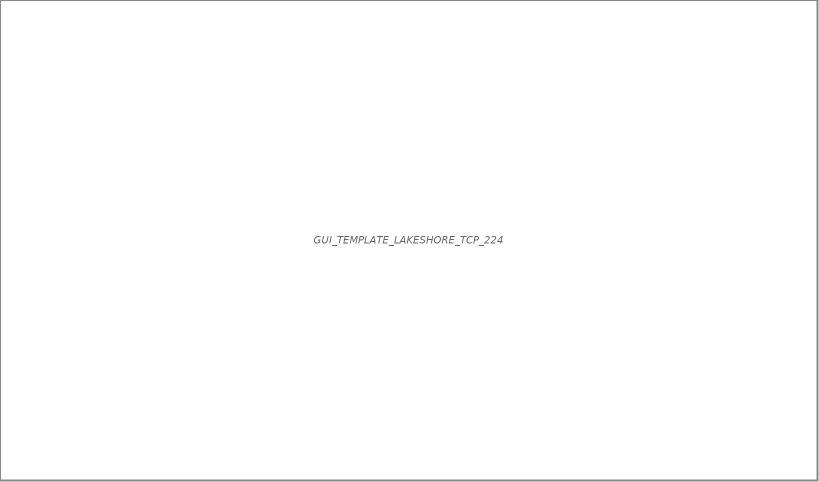
VISUALIZATION GUI_LAKESHORE_TCP_224_SIM  // 819x482
    Frame (0,0 817x480)
        shows GUI_TEMPLATE_LAKESHORE_TCP_224(m_Instance := MAIN.LS224_TCP_SIM)
END_VISUALIZATION

(* stored: Version 1.1.0.1, ProductVersion 3.1.4022.16
   Visu GUI_LAKESHORE_TCP_224_SIM: Id {3e6fd5e0-54a1-4676-a8a0-fb4aeefd8c6e} *)
